(* LS Electric XG5000 project: e_pcmaster_elec_room_controll *)
(* 전기실 환기제어 시스템 실제 적용 시스 템 및 지하주차장 환기 시스탬 *)
(* PLC LSPLC *)
(* module base 0 slot 0: 입출력 모듈:XBC-DR40S (DC 24V 입력 24점, 릴레이 출력 16점) *)
(* module base 0 slot 1: 온도입력 모듈:XBF-RD04A (RTD 온도 입력형 4채널) *)
(* module base 0 slot 2: 아날로그입력 모듈:XBF-AD04A (A/D 전압 전류 입력형 4채널) *)
(* task init: Kind=1 Priority=2 *)
VAR_GLOBAL
    autumn_set_sw : BIT; (* 가을철 온도 *)
    C1_B1_E_FR01_out : BIT;
    C1_B1_E_FR01_start_tk4s_set : WORD;
    C1_B1_E_FR02_out : BIT;
    C1_B1_E_FR02_start_tk4s_set : WORD;
    C1_B1_E_FR05_out : BIT;
    C1_B1_E_FR05_start_tk4s_set : WORD;
    C1_B1_E_FR06_out : BIT;
    C1_B1_E_FR06_start_tk4s_set : WORD;
    C1_B1_E_FR10_out : BIT;
    C1_B1_E_FR10_start_tk4s_set : WORD;
    C1_B1_S_FR03_out : BIT;
    C1_B1_S_FR03_select AT D06230.0 : BIT;
    C1_B1_S_FR03_start_tk4s_alarm_set : WORD;
    C1_B1_S_FR03_temp : WORD;
    C1_B1_S_FR04_out : BIT;
    C1_B1_S_FR04_select AT D06230.1 : BIT;
    C1_B1_S_FR04_start_tk4s_alarm_set : WORD;
    C1_B1_S_FR04_temp : WORD;
    C1_B1_S_FR07_out : BIT;
    C1_B1_S_FR07_select AT D06230.2 : BIT;
    C1_B1_S_FR07_start_tk4s_alarm_set : WORD;
    C1_B1_S_FR07_temp : WORD;
    C1_B1_S_FR08_out : BIT;
    C1_B1_S_FR08_select AT D06230.3 : BIT;
    C1_B1_S_FR08_start_tk4s_alarm_set : WORD;
    C1_B1_S_FR08_temp : WORD;
    C1_B1_S_FR09_out : BIT;
    C1_B1_S_FR09_select AT D06230.4 : BIT;
    C1_B1_S_FR09_start_tk4s_alarm_set : WORD;
    C1_B1_S_FR09_temp : WORD;
    C1_B2_E_FR01_out : BIT;
    C1_B2_E_FR01_start_tk4s_set : WORD;
    C1_B2_E_FR02_out : BIT;
    C1_B2_E_FR02_start_tk4s_set : WORD;
    C1_B2_E_FR05_out : BIT;
    C1_B2_E_FR05_start_tk4s_set : WORD;
    C1_B2_E_FR06_out : BIT;
    C1_B2_E_FR06_start_tk4s_set : WORD;
    C1_B2_E_FR10_out : BIT;
    C1_B2_E_FR10_start_tk4s_set : WORD;
    C1_B2_S_FR03_out : BIT;
    C1_B2_S_FR03_select AT D06230.5 : BIT;
    C1_B2_S_FR03_start_tk4s_alarm_set : WORD;
    C1_B2_S_FR03_temp : WORD;
    C1_B2_S_FR04_out : BIT;
    C1_B2_S_FR04_select AT D06230.6 : BIT;
    C1_B2_S_FR04_start_tk4s_alarm_set : WORD;
    C1_B2_S_FR04_temp : WORD;
    C1_B2_S_FR07_out : BIT;
    C1_B2_S_FR07_select AT D06230.7 : BIT;
    C1_B2_S_FR07_start_tk4s_alarm_set : WORD;
    C1_B2_S_FR07_temp : WORD;
    C1_B2_S_FR08_out : BIT;
    C1_B2_S_FR08_select AT D06230.8 : BIT;
    C1_B2_S_FR08_start_tk4s_alarm_set : WORD;
    C1_B2_S_FR08_temp : WORD;
    C1_B2_S_FR09_out : BIT;
    C1_B2_S_FR09_select AT D06230.9 : BIT;
    C1_B2_S_FR09_start_tk4s_alarm_set : WORD;
    C1_B2_S_FR09_temp : WORD;
    C2_B1_E_FR11_out : BIT;
    C2_B1_E_FR11_start_tk4s_set : WORD;
    C2_B1_S_FR12_out : BIT;
    C2_B1_S_FR12_select AT D06230.A : BIT;
    C2_B1_S_FR12_start_tk4s_alarm_set : WORD;
    C2_B1_S_FR12_temp : WORD;
    C2_B2_E_FR11_out : BIT;
    C2_B2_E_FR11_start_tk4s_set : WORD;
    C2_B2_S_FR12_out : BIT;
    C2_B2_S_FR12_select AT D06230.B : BIT;
    C2_B2_S_FR12_start_tk4s_alarm_set : WORD;
    C2_B2_S_FR12_temp : WORD;
    C2_B3_E_FR11_out : BIT;
    C2_B3_E_FR11_start_tk4s_set : WORD;
    C2_B3_S_FR12_out : BIT;
    C2_B3_S_FR12_select AT D06230.C : BIT;
    C2_B3_S_FR12_start_tk4s_alarm_set : WORD;
    C2_B3_S_FR12_temp : WORD;
    cold_winter_set_sw : BIT;
    early_winter_set_sw : BIT; (* 초겨울 *)
    EF_operation AT M00203 : BIT;
    heart_beat_manual_sw : BIT;
    heart_beat_mem : WORD;
    heart_beat_timer : TIMER;
    Park_1H_time : WORD;
    Park_auto_B_manual_A : BIT;
    Park_auto_start : BIT;
    Park_daily_schedule_on : BIT;
    Park_manual_cont_ind_start : BIT;
    Park_manual_cont_tot_start : BIT;
    Park_manual_con_B_time_A : BIT;
    Park_manual_ind_B_tot_A : BIT;
    Park_manual_ind_start_out : BIT;
    Park_manual_oper_time : WORD;
    Park_manual_start : BIT;
    Park_manual_timer : TIMER;
    Park_manual_time_ind_start : BIT;
    Park_manual_time_tot_start : BIT;
    Park_manual_total_start_out : BIT;
    Park_manual_순차가동_2R : DWORD;
    Park_manual_순차기동_계산값 : WORD;
    Park_manual_순차기동_전송값 : WORD;
    Park_schedule_06_start : BIT;
    Park_schedule_08_start : BIT;
    Park_schedule_09_start : BIT;
    Park_schedule_10_start : BIT;
    Park_schedule_15_stop : BIT;
    Park_schedule_17stop : BIT;
    Park_schedule_18stop : BIT;
    Park_schedule_20stop : BIT;
    Park_schedule_autumn : BIT;
    Park_schedule_spring : BIT;
    Park_schedule_summer : BIT;
    Park_schedule_winter : BIT;
    Park_start_B_stop_A : BIT;
    Park_temp_1_high : WORD;
    Park_temp_1_high_H_set : WORD;
    Park_temp_1_high_L_set : WORD;
    Park_temp_2_med_high : WORD;
    Park_temp_2_med_high_H_set : WORD;
    Park_temp_2_med_high_L_set : WORD;
    Park_temp_3_med : WORD;
    Park_temp_3_med_H_set : WORD;
    Park_temp_3_med_L_set : WORD;
    Park_temp_4_med_low : WORD;
    Park_temp_4_med_low_H_set : WORD;
    Park_temp_4_med_low_L_set : WORD;
    Park_temp_5_low : WORD;
    Park_temp_5_low_H_set : WORD;
    Park_temp_5_low_L_set : WORD;
    Park_temp_6_low_1 : WORD;
    Park_temp_6_low_1_oper_time : WORD;
    Park_temp_7_low_2 : WORD;
    Park_temp_7_low_2_oper_time : WORD;
    Park_temp_8_low_3 : WORD;
    Park_temp_8_low_3_oper_time : WORD;
    Park_temp_9_below0 : WORD;
    Park_temp_9_below0_oper_time : WORD;
    Park_time_oper_delay_time : WORD;
    Park_tk4m_alarm_start_set : WORD;
    Park_tk4m_alarm_stop_set : WORD;
    Park_tk4m_start_set : WORD;
    Park_tk4m_stop_set : WORD;
    Park_순차기동_카운터 : COUNTER;
    Park_순차기동_타이머 : TIMER;
    SF_operation AT M00209 : BIT;
    spring_set_sw : BIT; (* spring_set_sw *)
    summer_set_sw : BIT; (* 하절기운전온도 변경 *)
    tr01_1m_high_temp_from_pc AT D00980 : WORD;
    tr01_temp_scaled_value AT D00024 : WORD;
    tr02_1m_high_temp_from_pc AT D00981 : WORD;
    tr02_temp_scaled_value AT D00025 : WORD;
    tr03_1m_high_temp_from_pc AT D00982 : WORD;
    tr03_temp_scaled_value AT D00026 : WORD;
    winter_set_sw : BIT; (* 겨울철 *)
    _002_1C_1B_FR01_temp : WORD; (* _002_1C_1B_FR01_temp *)
    _002_1C_1B_FR02_temp : WORD; (* _002_1C_1B_FR02_temp *)
    _002_1C_1B_FR03_temp : WORD; (* _002_1C_1B_FR03_temp *)
    _002_1C_1B_FR04_temp : WORD; (* _002_1C_1B_FR04_temp *)
    _002_1C_1B_FR05_temp : WORD; (* _002_1C_1B_FR05_temp *)
    _002_1C_2B_FR01_temp : WORD; (* _002_1C_2B_FR01_temp *)
    _002_1C_2B_FR02_temp : WORD; (* _002_1C_2B_FR02_temp *)
    _002_1C_2B_FR03_temp : WORD; (* _002_1C_2B_FR03_temp *)
    _002_1C_2B_FR04_temp : WORD; (* _002_1C_2B_FR04_temp *)
    _002_1C_2B_FR05_temp : WORD; (* _002_1C_2B_FR05_temp *)
    _002_tr_1_temp : WORD; (* _002_tr_1_temp *)
    _002_tr_2_temp : WORD; (* _002_tr_2_temp *)
    _002_tr_3_temp : WORD; (* _002_tr_3_temp *)
    _002_W_011_reserved : WORD; (* _002_W_011_reserved *)
    _002_W_012_reserved : WORD; (* _002_W_012_reserved *)
    _003_tr_1_AB_valtage : DWORD; (* _003_tr_1_AB_valtage *)
    _003_tr_1_A_current : DWORD; (* _003_tr_1_A_current *)
    _003_tr_1_A_valtage : DWORD; (* _003_tr_1_A_valtage *)
    _003_tr_1_BC_valtage : DWORD; (* _003_tr_1_BC_valtage *)
    _003_tr_1_B_current : DWORD; (* _003_tr_1_B_current *)
    _003_tr_1_B_valtage : DWORD; (* _003_tr_1_B_valtage *)
    _003_tr_1_CA_valtage : DWORD; (* _003_tr_1_CA_valtage *)
    _003_tr_1_C_current : DWORD; (* _003_tr_1_C_current *)
    _003_tr_1_C_valtage : DWORD; (* _003_tr_1_C_valtage *)
    _003_tr_1_effective_power : DWORD; (* _003_tr_1_effective_power *)
    _003_tr_1_power : DWORD; (* _003_tr_1_power *)
    _003_tr_1_power_factor : DWORD; (* _003_tr_1_power_factor *)
    _003_tr_1_reactive_power : DWORD; (* _003_tr_1_reactive_power *)
    _004_tr_2_AB_valtage : DWORD; (* _004_tr_2_AB_valtage *)
    _004_tr_2_A_current : DWORD; (* _004_tr_2_A_current *)
    _004_tr_2_A_valtage : DWORD; (* _004_tr_2_A_valtage *)
    _004_tr_2_BC_valtage : DWORD; (* _004_tr_2_BC_valtage *)
    _004_tr_2_B_current : DWORD; (* _004_tr_2_B_current *)
    _004_tr_2_B_valtage : DWORD; (* _004_tr_2_B_valtage *)
    _004_tr_2_CA_valtage : DWORD; (* _004_tr_2_CA_valtage *)
    _004_tr_2_C_current : DWORD; (* _004_tr_2_C_current *)
    _004_tr_2_C_valtage : DWORD; (* _004_tr_2_C_valtage *)
    _004_tr_2_effective_power : DWORD; (* _004_tr_2_effective_power *)
    _004_tr_2_power : DWORD; (* _004_tr_2_power *)
    _004_tr_2_power_factor : DWORD; (* _004_tr_2_power_factor *)
    _004_tr_2_reactive_power : DWORD; (* _004_tr_2_reactive_power *)
    _005_tr_3_AB_valtage : DWORD; (* _005_tr_3_AB_valtage *)
    _005_tr_3_A_current : DWORD; (* _005_tr_3_A_current *)
    _005_tr_3_A_valtage : DWORD; (* _005_tr_3_A_valtage *)
    _005_tr_3_BC_valtage : DWORD; (* _005_tr_3_BC_valtage *)
    _005_tr_3_B_current : DWORD; (* _005_tr_3_B_current *)
    _005_tr_3_B_valtage : DWORD; (* _005_tr_3_B_valtage *)
    _005_tr_3_CA_valtage : DWORD; (* _005_tr_3_CA_valtage *)
    _005_tr_3_C_current : DWORD; (* _005_tr_3_C_current *)
    _005_tr_3_C_valtage : DWORD; (* _005_tr_3_C_valtage *)
    _005_tr_3_effective_power : DWORD; (* _005_tr_3_effective_power *)
    _005_tr_3_power : DWORD; (* _005_tr_3_power *)
    _005_tr_3_power_factor : DWORD; (* _005_tr_3_power_factor *)
    _005_tr_3_reactive_power : DWORD; (* _005_tr_3_reactive_power *)
    _007_outdoor_temp : WORD; (* _007_outdoor_temp *)
    _007_room_temp : WORD; (* _007_room_temp *)
    _008_room_temp_high_set AT D00906 : WORD; (* _008_room_temp_high_set *)
    _008_room_temp_high_set_high_limit : WORD; (* _008_room_temp_high_set_high_limit *)
    _008_room_temp_high_set_low_limit : WORD; (* _008_room_temp_high_set_low_limit *)
    _008_room_temp_low_set AT D00907 : WORD; (* _008_room_temp_low_set *)
    _008_room_temp_low_set_high_limit : WORD; (* _008_room_temp_low_set_high_limit *)
    _008_room_temp_low_set_low_limit : WORD; (* _008_room_temp_low_set_low_limit *)
    _009_outdoor_temp_high_set AT D00908 : WORD; (* _009_outdoor_temp_high_set *)
    _009_outdoor_temp_high_set_high_limit : WORD; (* _009_outdoor_temp_high_set_high_limit *)
    _009_outdoor_temp_high_set_low_limit : WORD; (* _009_outdoor_temp_high_set_low_limit *)
    _009_outdoor_temp_low_set AT D00909 : WORD; (* _009_outdoor_temp_low_set *)
    _009_outdoor_temp_low_set_high_limit : WORD; (* _009_outdoor_temp_low_set_high_limit *)
    _009_outdoor_temp_low_set_low_limit : WORD; (* _009_outdoor_temp_low_set_low_limit *)
    _010_D_00 : DWORD; (* _010_D_00 *)
    _010_D_01 : DWORD; (* _010_D_01 *)
    _010_D_unit_hour_cost : DWORD; (* _010_D_unit_hour_cost *)
    _010_R_00 : DWORD; (* _010_R_00 *)
    _010_R_01 : DWORD; (* _010_R_01 *)
    _010_R_power_unit_price_percent : DWORD; (* _010_R_power_unit_price_percent *)
    _010_R_unit_hour_cost : DWORD; (* _010_R_unit_hour_cost *)
    _010_W_02 : WORD; (* _010_W_02 *)
    _010_W_03 : WORD; (* _010_W_03 *)
    _010_W_1hr_count : WORD; (* _010_W_1hr_count *)
    _010_W_1_thousand_hour : WORD; (* _010_W_1_thousand_hour *)
    _010_W_fan_power_capacity : WORD; (* _010_W_fan_power_capacity *)
    _010_W_high_low_diff : WORD; (* _010_W_high_low_diff *)
    _010_W_power_unit_price : WORD; (* _010_W_power_unit_price *)
    _010_W_TR1_temp_high_set AT D00900 : WORD;
    _010_W_TR1_temp_low_set AT D00901 : WORD;
    _010_W_TR2_temp_high_set AT D00902 : WORD;
    _010_W_TR2_temp_low_set AT D00903 : WORD;
    _010_W_TR3_temp_high_set AT D00904 : WORD; (* _010_W_TR_temp_high_set *)
    _010_W_TR3_temp_low_set AT D00905 : WORD; (* _010_W_TR_temp_low_set *)
    _01_CH0_TEMP AT U01.04 : WORD; (* 온도입력모듈 : 채널0 온도변환값(전기실온도) *)
    _01_CH1_TEMP AT U01.05 : WORD; (* 온도입력모듈 : 채널1 온도변환값(외기온도) *)
    _01_CH2_TEMP AT U01.06 : WORD; (* 온도입력모듈 : 채널2 온도변환값(에어콘01출구온도) *)
    _01_CH3_TEMP AT U01.07 : WORD; (* 온도입력모듈 : 채널3 온도변환값(에어콘02출구온도) *)
    _02_CH0_DATA AT U02.02 : WORD; (* 아날로그입력 모듈: 채널0 변환값(tr01 temp) *)
    _02_CH1_DATA AT U02.03 : WORD; (* 아날로그입력 모듈: 채널1 변환값(tr02 temp) *)
    _02_CH2_DATA AT U02.04 : WORD; (* 아날로그입력 모듈: 채널2 변환값(tr01 temp) *)
    _IC_1B_FR01_temp_high_set : BIT;
    _주차장_급기팬_가동 : BIT;
    _주차장_급기팬_정지 : BIT;
    월간타이머리셋 : BIT;
    전기실_급배기_동시기동방지 : TIMER; (* 전기실_급배기_동시기동방지 *)
    주차장_급기가동온도 : WORD;
    주차장_급기정지온도 : WORD; (* 주차장_제어_외기_고온도 *)
END_VAR
VAR_GLOBAL RETAIN
    Park_oper_time_add : WORD;
    TR1_opertime_time : WORD;
    TR1_opertime_timer : TIMER;
    TR2_opertime_time : WORD;
    TR2_opertime_timer : TIMER;
    TR3_opertime_time : WORD;
    TR3_opertime_timer : TIMER;
    TR_opertime_total_time : WORD;
    _000_EF_tot_local_auto_op_timer : TIMER; (* _000_EF_tot_local_auto_op_timer *)
    _000_EF_tot_local_manual_op_timer : TIMER; (* _000_EF_tot_local_manual_op_timer *)
    _000_EF_tot_op_room_op_timer : TIMER; (* _000_EF_tot_op_room_op_timer *)
    _000_EF_tot_op_timer : TIMER; (* _000_EF_tot_op_timer *)
    _000_SF_tot_local_auto_op_timer : TIMER; (* _000_SF_tot_local_auto_op_timer *)
    _000_SF_tot_local_manual_op_timer : TIMER; (* _000_SF_tot_local_manual_op_timer *)
    _000_SF_tot_op_room_op_timer : TIMER; (* _000_SF_tot_op_room_op_timer *)
    _000_SF_tot_op_timer : TIMER; (* _000_SF_tot_op_timer *)
    _001_EF_tot_local_auto_op_hour : WORD; (* _001_EF_tot_local_auto_op_hour *)
    _001_EF_tot_local_manual_op_hour : WORD; (* _001_EF_tot_local_manual_op_hour *)
    _001_EF_tot_op_hour : WORD; (* _001_EF_tot_op_hour *)
    _001_EF_tot_op_room_op_hour : WORD; (* _001_EF_tot_op_room_op_hour *)
    _001_SF_tot_local_auto_op_hour : WORD; (* _001_SF_tot_local_auto_op_hour *)
    _001_SF_tot_local_manual_op_hour : WORD; (* _001_SF_tot_local_manual_op_hour *)
    _001_SF_tot_op_hour : WORD; (* _001_SF_tot_op_hour *)
    _001_SF_tot_op_room_op_hour : WORD; (* _001_SF_tot_op_room_op_hour *)
    _001_tot_local_auto_op_hour : WORD; (* _001_tot_local_auto_op_hour *)
    _001_tot_local_manual_op_hour : WORD; (* _001_tot_local_manual_op_hour *)
    _001_tot_op_hour : WORD; (* _001_tot_op_hour *)
    _001_tot_op_room_op_hour : WORD; (* _001_tot_op_room_op_hour *)
    _006_EF_tot_local_auto_op_hour : COUNTER; (* _006_EF_tot_local_auto_op_hour *)
    _006_EF_tot_local_manual_op_hour : COUNTER; (* _006_EF_tot_local_manual_op_hour *)
    _006_EF_tot_op_hour : COUNTER; (* _006_ESF_tot_op_hour *)
    _006_EF_tot_op_room_op_hour : COUNTER; (* _006_EF_tot_op_room_op_hour *)
    _006_SF_tot_local_auto_op_hour : COUNTER; (* _006_SF_tot_local_auto_op_hour *)
    _006_SF_tot_local_manual_op_hour : COUNTER; (* _006_SF_tot_local_manual_op_hour *)
    _006_SF_tot_op_hour : COUNTER; (* _006_SF_tot_op_hour *)
    _006_SF_tot_op_room_op_hour : COUNTER; (* _006_SF_tot_op_room_op_hour *)
END_VAR

PROGRAM elec_room_ventilation (* task: 스캔 프로그램 *)
VAR
    aircon01_operation AT M00221 : BIT;
    aircon01_OP_value AT D00957 : WORD;
    aircon02_operation AT M00222 : BIT;
    aircon02_OP_value AT D00958 : WORD;
    aircon_operation : BIT;
    basic_win_2_main_menu : BIT; (* basic_win_2_main_menu *)
    basic_win_2_main_menu_action : BIT; (* basic_win_2_main_menu_action *)
    basic_win_3_main_menu : BIT; (* basic_win_3_main_menu *)
    basic_win_3_main_menu_action : BIT; (* basic_win_3_main_menu_action *)
    basic_win_5_main_menu : BIT; (* basic_win_5_main_menu *)
    basic_win_5_main_menu_action : BIT; (* basic_win_5_main_menu_action *)
    EF_local_auto_start AT M00105 : BIT; (* EF_local_auto_start *)
    EF_local_auto_start_out AT M00200 : BIT; (* EF_local_auto_start_out *)
    EF_local_manual_start AT M00106 : BIT; (* EF_local_manual_start *)
    EF_local_manual_start_out AT M00201 : BIT; (* EF_local_manual_start_out *)
    EF_local_manual_start_sw AT M00116 : BIT; (* EF_local_manual_start_sw *)
    EF_op_room_start AT M00107 : BIT; (* EF_op_room_start *)
    EF_op_room_start_out AT M00202 : BIT; (* EF_op_room_start_out *)
    EF_stop AT M00108 : BIT; (* EF_stop *)
    EF_stop_out AT M00204 : BIT; (* EF_stop_out *)
    EF_trip AT M00205 : BIT; (* EF_trip *)
    EF_trip_reset AT M00109 : BIT; (* EF_trip_reset *)
    outdoor_temp_high_set_sw : BIT; (* outdoor_temp_high_set_sw *)
    outdoor_temp_low_set_sw : BIT; (* outdoor_temp_low_set_sw *)
    plc_error : BIT;
    plc_run : BIT;
    room_temp_high_set_sw : BIT; (* room_temp_high_set_sw *)
    room_temp_low_set_sw : BIT; (* room_temp_low_set_sw *)
    room_temp_trend_win_open : BIT; (* room_temp_trend_win_open *)
    room_temp_trend_win_trigger : BIT; (* room_temp_trend_win_trigger *)
    SF_local_auto_point_hour : BIT; (* SF_local_auto_point_hour *)
    SF_local_auto_start AT M00110 : BIT; (* SF_local_auto_start *)
    SF_local_auto_start_out AT M00206 : BIT; (* SF_local_auto_start_out *)
    SF_local_manual_point_hour : BIT; (* SF_local_manual_point_hour *)
    SF_local_manual_start AT M00111 : BIT; (* SF_local_manual_start *)
    SF_local_manual_start_out AT M00207 : BIT; (* SF_local_manual_start_out *)
    SF_local_manual_start_sw AT M00117 : BIT; (* SF_local_manual_start_sw *)
    SF_op_room_point_hour : BIT; (* SF_op_room_point_hour *)
    SF_op_room_start AT M00112 : BIT; (* SF_op_room_start *)
    SF_op_room_start_out AT M00208 : BIT; (* SF_op_room_start_out *)
    SF_stop AT M00113 : BIT; (* SF_stop *)
    SF_stop_out AT M00210 : BIT; (* SF_stop_out *)
    SF_tot_point_hour : BIT; (* SF_tot_point_hour *)
    sf_trip AT M00211 : BIT; (* sf_trip *)
    SF_trip_reset AT M00114 : BIT; (* SF_trip_reset *)
    tr_temp_trend_win_open : BIT; (* tr_temp_trend_win_open *)
    tr_temp_trend_win_trigger : BIT; (* tr_temp_trend_win_trigger *)
    unit_price_change : BIT; (* unit_price_change *)
    unit_price_change_action : BIT; (* unit_price_change_action *)
    unit_price_change_complete : BIT; (* unit_price_change_complete *)
    unit_price_change_complete_action : BIT; (* unit_price_change_complete_action *)
    unit_price_change_password : WORD; (* unit_price_change_password *)
    unit_price_change_password_fail : BIT; (* unit_price_change_password_fail *)
    unit_price_change_password_ok : BIT; (* unit_price_change_password_ok *)
    unit_price_change_pw_fail : BIT; (* unit_price_change_pw_fail *)
    unit_price_change_pw_ok : BIT; (* unit_price_change_pw_ok *)
    unit_price_change_temp_value : WORD; (* unit_price_change_temp_value *)
    win_2_view_graph : BIT; (* win_2_view_graph *)
    win_2_view_graph_open : BIT; (* win_2_view_graph_open *)
    _007_outdoor_temp_max_reset : BIT;
END_VAR
VAR_EXTERNAL
    autumn_set_sw : BIT; (* 가을철 온도 *)
    EF_operation : BIT; (* AT M00203 *)
    heart_beat_manual_sw : BIT;
    heart_beat_mem : WORD;
    heart_beat_timer : TIMER;
    SF_operation : BIT; (* AT M00209 *)
    tr01_1m_high_temp_from_pc : WORD; (* AT D00980 *)
    tr01_temp_scaled_value : WORD; (* AT D00024 *)
    tr02_1m_high_temp_from_pc : WORD; (* AT D00981 *)
    tr02_temp_scaled_value : WORD; (* AT D00025 *)
    tr03_1m_high_temp_from_pc : WORD; (* AT D00982 *)
    tr03_temp_scaled_value : WORD; (* AT D00026 *)
    winter_set_sw : BIT; (* 겨울철 *)
    _007_outdoor_temp : WORD; (* _007_outdoor_temp *)
    _007_room_temp : WORD; (* _007_room_temp *)
    _008_room_temp_high_set : WORD; (* AT D00906 *) (* _008_room_temp_high_set *)
    _008_room_temp_high_set_high_limit : WORD; (* _008_room_temp_high_set_high_limit *)
    _008_room_temp_high_set_low_limit : WORD; (* _008_room_temp_high_set_low_limit *)
    _008_room_temp_low_set : WORD; (* AT D00907 *) (* _008_room_temp_low_set *)
    _008_room_temp_low_set_high_limit : WORD; (* _008_room_temp_low_set_high_limit *)
    _008_room_temp_low_set_low_limit : WORD; (* _008_room_temp_low_set_low_limit *)
    _009_outdoor_temp_high_set : WORD; (* AT D00908 *) (* _009_outdoor_temp_high_set *)
    _009_outdoor_temp_low_set : WORD; (* AT D00909 *) (* _009_outdoor_temp_low_set *)
    _010_W_power_unit_price : WORD; (* _010_W_power_unit_price *)
    _01_CH0_TEMP : WORD; (* AT U01.04 *) (* 온도입력모듈 : 채널0 온도변환값(전기실온도) *)
    _01_CH1_TEMP : WORD; (* AT U01.05 *) (* 온도입력모듈 : 채널1 온도변환값(외기온도) *)
    월간타이머리셋 : BIT;
    전기실_급배기_동시기동방지 : TIMER; (* 전기실_급배기_동시기동방지 *)
END_VAR

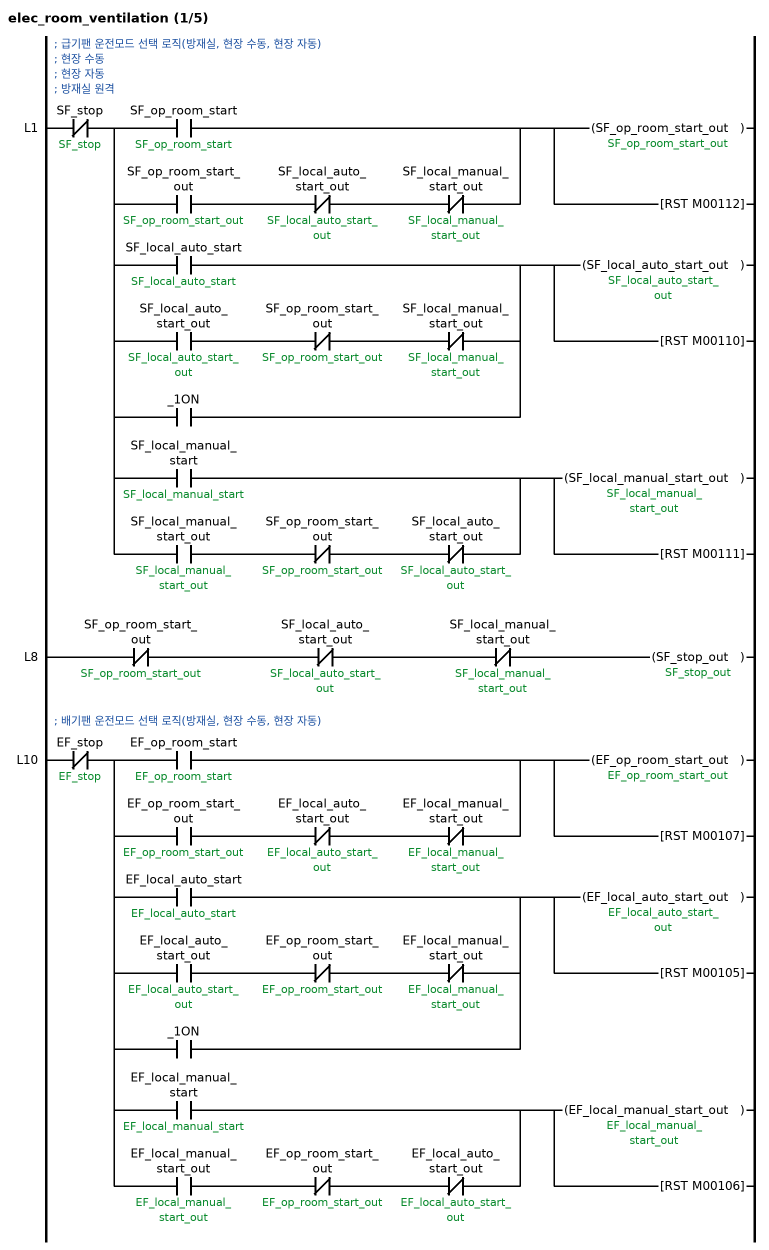
// 급기팬 운전모드 선택 로직(방재실, 현장 수동, 현장 자동)
; L1
LOAD NOT  SF_stop	// SF_stop
MPUSH
LOAD      SF_op_room_start	// SF_op_room_start
LOAD      SF_op_room_start_out	// SF_op_room_start_out
AND NOT   SF_local_auto_start_out	// SF_local_auto_start_out
AND NOT   SF_local_manual_start_out	// SF_local_manual_start_out
OR LOAD
AND LOAD
OUT       SF_op_room_start_out	// SF_op_room_start_out
RST       M00112
MLOAD
LOAD      SF_local_auto_start	// SF_local_auto_start
LOAD      SF_local_auto_start_out	// SF_local_auto_start_out
AND NOT   SF_op_room_start_out	// SF_op_room_start_out
AND NOT   SF_local_manual_start_out	// SF_local_manual_start_out
OR LOAD
OR        _1ON
AND LOAD
OUT       SF_local_auto_start_out	// SF_local_auto_start_out
RST       M00110
MPOP
LOAD      SF_local_manual_start	// SF_local_manual_start
LOAD      SF_local_manual_start_out	// SF_local_manual_start_out
AND NOT   SF_op_room_start_out	// SF_op_room_start_out
AND NOT   SF_local_auto_start_out	// SF_local_auto_start_out
OR LOAD
AND LOAD
OUT       SF_local_manual_start_out	// SF_local_manual_start_out
RST       M00111
// output comment: 현장 수동
// output comment: 현장 자동
// output comment: 방재실 원격
; L8
LOAD NOT  SF_op_room_start_out	// SF_op_room_start_out
AND NOT   SF_local_auto_start_out	// SF_local_auto_start_out
AND NOT   SF_local_manual_start_out	// SF_local_manual_start_out
OUT       SF_stop_out	// SF_stop_out
// 배기팬 운전모드 선택 로직(방재실, 현장 수동, 현장 자동)
; L10
LOAD NOT  EF_stop	// EF_stop
MPUSH
LOAD      EF_op_room_start	// EF_op_room_start
LOAD      EF_op_room_start_out	// EF_op_room_start_out
AND NOT   EF_local_auto_start_out	// EF_local_auto_start_out
AND NOT   EF_local_manual_start_out	// EF_local_manual_start_out
OR LOAD
AND LOAD
OUT       EF_op_room_start_out	// EF_op_room_start_out
RST       M00107
MLOAD
LOAD      EF_local_auto_start	// EF_local_auto_start
LOAD      EF_local_auto_start_out	// EF_local_auto_start_out
AND NOT   EF_op_room_start_out	// EF_op_room_start_out
AND NOT   EF_local_manual_start_out	// EF_local_manual_start_out
OR LOAD
OR        _1ON
AND LOAD
OUT       EF_local_auto_start_out	// EF_local_auto_start_out
RST       M00105
MPOP
LOAD      EF_local_manual_start	// EF_local_manual_start
LOAD      EF_local_manual_start_out	// EF_local_manual_start_out
AND NOT   EF_op_room_start_out	// EF_op_room_start_out
AND NOT   EF_local_auto_start_out	// EF_local_auto_start_out
OR LOAD
AND LOAD
OUT       EF_local_manual_start_out	// EF_local_manual_start_out
RST       M00106

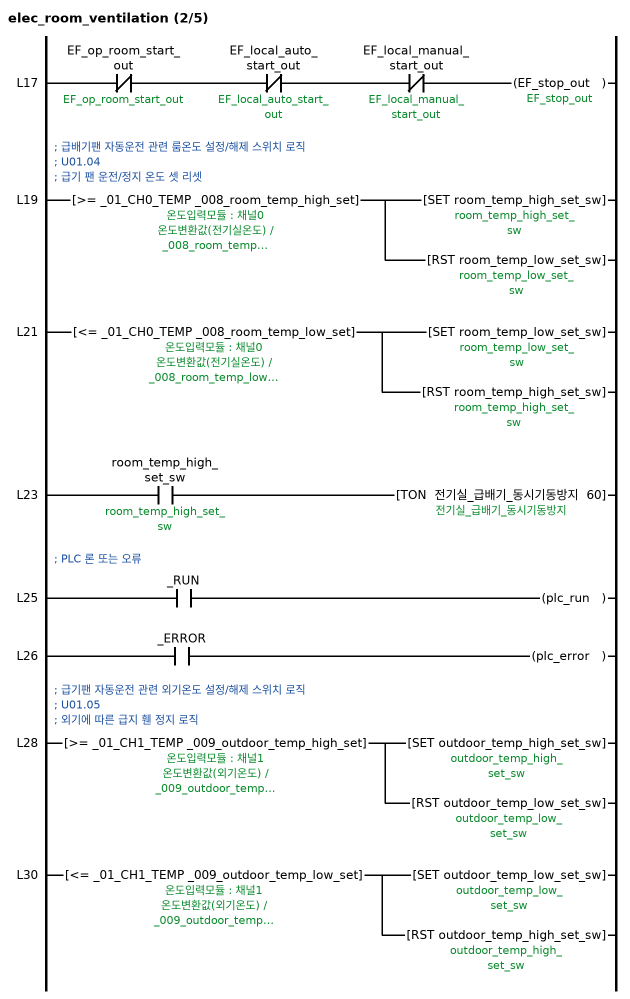
; L17
LOAD NOT  EF_op_room_start_out	// EF_op_room_start_out
AND NOT   EF_local_auto_start_out	// EF_local_auto_start_out
AND NOT   EF_local_manual_start_out	// EF_local_manual_start_out
OUT       EF_stop_out	// EF_stop_out
// 급배기팬 자동운전 관련 룸온도 설정/해제 스위치 로직
; L19
LOAD>=    _01_CH0_TEMP _008_room_temp_high_set	// 온도입력모듈 : 채널0 온도변환값(전기실온도) / _008_room_temp_high_set
SET       room_temp_high_set_sw	// room_temp_high_set_sw
RST       room_temp_low_set_sw	// room_temp_low_set_sw
// output comment: U01.04
// output comment: 급기 팬 운전/정지 온도 셋 리셋
; L21
LOAD<=    _01_CH0_TEMP _008_room_temp_low_set	// 온도입력모듈 : 채널0 온도변환값(전기실온도) / _008_room_temp_low_set
SET       room_temp_low_set_sw	// room_temp_low_set_sw
RST       room_temp_high_set_sw	// room_temp_high_set_sw
; L23
LOAD      room_temp_high_set_sw	// room_temp_high_set_sw
TON       전기실_급배기_동시기동방지 60	// 전기실_급배기_동시기동방지
// PLC 론 또는 오류
; L25
LOAD      _RUN
OUT       plc_run
; L26
LOAD      _ERROR
OUT       plc_error
// 급기팬 자동운전 관련 외기온도 설정/해제 스위치 로직
; L28
LOAD>=    _01_CH1_TEMP _009_outdoor_temp_high_set	// 온도입력모듈 : 채널1 온도변환값(외기온도) / _009_outdoor_temp_high_set
SET       outdoor_temp_high_set_sw	// outdoor_temp_high_set_sw
RST       outdoor_temp_low_set_sw	// outdoor_temp_low_set_sw
// output comment: U01.05
// output comment: 외기에 따른 급지 휀 정지 로직
; L30
LOAD<=    _01_CH1_TEMP _009_outdoor_temp_low_set	// 온도입력모듈 : 채널1 온도변환값(외기온도) / _009_outdoor_temp_low_set
SET       outdoor_temp_low_set_sw	// outdoor_temp_low_set_sw
RST       outdoor_temp_high_set_sw	// outdoor_temp_high_set_sw

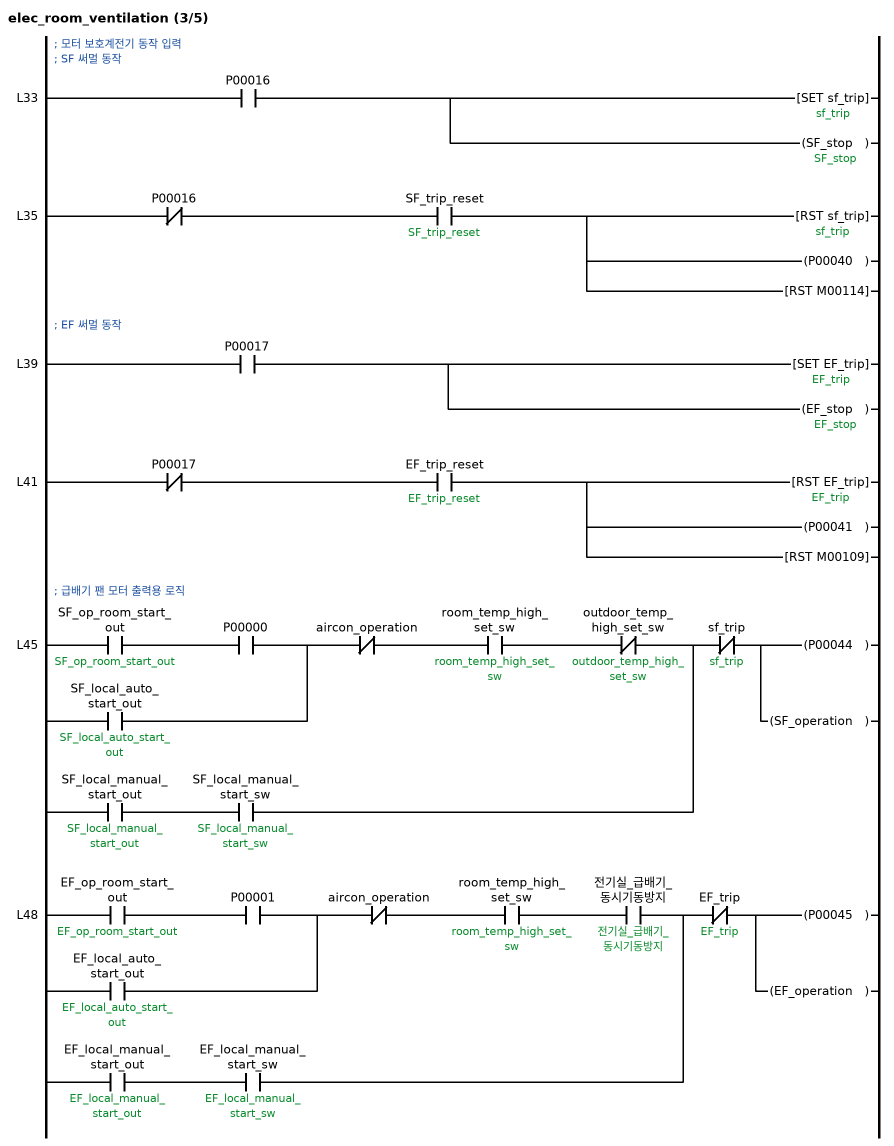
// 모터 보호계전기 동작 입력
; L33
LOAD      P00016
SET       sf_trip	// sf_trip
OUT       SF_stop	// SF_stop
// output comment: SF 써멀 동작
; L35
LOAD NOT  P00016
AND       SF_trip_reset	// SF_trip_reset
RST       sf_trip	// sf_trip
OUT       P00040
RST       M00114
; L39
LOAD      P00017
SET       EF_trip	// EF_trip
OUT       EF_stop	// EF_stop
// output comment: EF 써멀 동작
; L41
LOAD NOT  P00017
AND       EF_trip_reset	// EF_trip_reset
RST       EF_trip	// EF_trip
OUT       P00041
RST       M00109
// 급배기 팬 모터 출력용 로직
; L45
LOAD      SF_op_room_start_out	// SF_op_room_start_out
AND       P00000
OR        SF_local_auto_start_out	// SF_local_auto_start_out
AND NOT   aircon_operation
AND       room_temp_high_set_sw	// room_temp_high_set_sw
AND NOT   outdoor_temp_high_set_sw	// outdoor_temp_high_set_sw
LOAD      SF_local_manual_start_out	// SF_local_manual_start_out
AND       SF_local_manual_start_sw	// SF_local_manual_start_sw
OR LOAD
AND NOT   sf_trip	// sf_trip
OUT       P00044
OUT       SF_operation
; L48
LOAD      EF_op_room_start_out	// EF_op_room_start_out
AND       P00001
OR        EF_local_auto_start_out	// EF_local_auto_start_out
AND NOT   aircon_operation
AND       room_temp_high_set_sw	// room_temp_high_set_sw
AND       전기실_급배기_동시기동방지	// 전기실_급배기_동시기동방지
LOAD      EF_local_manual_start_out	// EF_local_manual_start_out
AND       EF_local_manual_start_sw	// EF_local_manual_start_sw
OR LOAD
AND NOT   EF_trip	// EF_trip
OUT       P00045
OUT       EF_operation

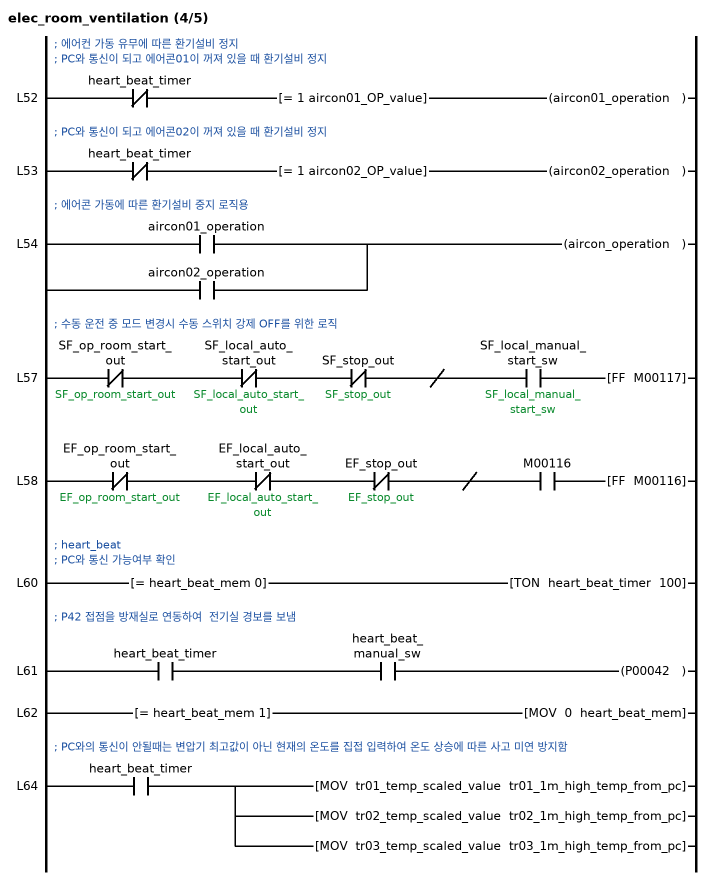
// 에어컨 가동 유무에 따른 환기설비 정지
; L52
LOAD NOT  heart_beat_timer
AND=      1 aircon01_OP_value
OUT       aircon01_operation
// output comment: PC와 통신이 되고 에어콘01이 꺼져 있을 때 환기설비 정지
; L53
LOAD NOT  heart_beat_timer
AND=      1 aircon02_OP_value
OUT       aircon02_operation
// output comment: PC와 통신이 되고 에어콘02이 꺼져 있을 때 환기설비 정지
; L54
LOAD      aircon01_operation
OR        aircon02_operation
OUT       aircon_operation
// output comment: 에어콘 가동에 따른 환기설비 중지 로직용
// 수동 운전 중 모드 변경시 수동 스위치 강제 OFF를 위한 로직
; L57
LOAD NOT  SF_op_room_start_out	// SF_op_room_start_out
AND NOT   SF_local_auto_start_out	// SF_local_auto_start_out
AND NOT   SF_stop_out	// SF_stop_out
NOT
AND       SF_local_manual_start_sw	// SF_local_manual_start_sw
FF        M00117
; L58
LOAD NOT  EF_op_room_start_out	// EF_op_room_start_out
AND NOT   EF_local_auto_start_out	// EF_local_auto_start_out
AND NOT   EF_stop_out	// EF_stop_out
NOT
AND       M00116
FF        M00116
// heart_beat
; L60
LOAD=     heart_beat_mem 0
TON       heart_beat_timer 100
// output comment: PC와 통신 가능여부 확인
; L61
LOAD      heart_beat_timer
AND       heart_beat_manual_sw
OUT       P00042
// output comment: P42 접점을 방재실로 연동하여  전기실 경보를 보냄
; L62
LOAD=     heart_beat_mem 1
MOV       0 heart_beat_mem
; L64
LOAD      heart_beat_timer
MOV       tr01_temp_scaled_value tr01_1m_high_temp_from_pc
MOV       tr02_temp_scaled_value tr02_1m_high_temp_from_pc
MOV       tr03_temp_scaled_value tr03_1m_high_temp_from_pc
// output comment: PC와의 통신이 안될때는 변압기 최고값이 아닌 현재의 온도를 집접 입력하여 온도 상승에 따른 사고 미연 방지함

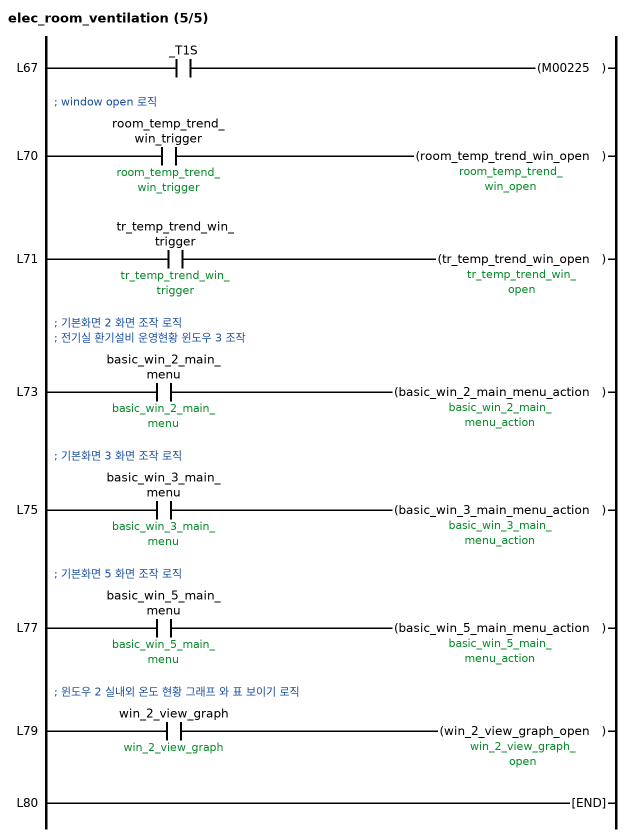
; L67
LOAD      _T1S
OUT       M00225
// window open 로직
; L70
LOAD      room_temp_trend_win_trigger	// room_temp_trend_win_trigger
OUT       room_temp_trend_win_open	// room_temp_trend_win_open
; L71
LOAD      tr_temp_trend_win_trigger	// tr_temp_trend_win_trigger
OUT       tr_temp_trend_win_open	// tr_temp_trend_win_open
// 기본화면 2 화면 조작 로직
; L73
LOAD      basic_win_2_main_menu	// basic_win_2_main_menu
OUT       basic_win_2_main_menu_action	// basic_win_2_main_menu_action
// output comment: 전기실 환기설비 운영현황 윈도우 3 조작
// 기본화면 3 화면 조작 로직
; L75
LOAD      basic_win_3_main_menu	// basic_win_3_main_menu
OUT       basic_win_3_main_menu_action	// basic_win_3_main_menu_action
// 기본화면 5 화면 조작 로직
; L77
LOAD      basic_win_5_main_menu	// basic_win_5_main_menu
OUT       basic_win_5_main_menu_action	// basic_win_5_main_menu_action
// 윈도우 2 실내외 온도 현황 그래프 와 표 보이기 로직
; L79
LOAD      win_2_view_graph	// win_2_view_graph
OUT       win_2_view_graph_open	// win_2_view_graph_open
; L80
END
END_PROGRAM

PROGRAM tr_cooling_logic (* task: 스캔 프로그램 *)
(* 온도 제어로 하절기 tr cooling fan 제어 *)
VAR
    temp_tr01_temp : WORD; (* temp_tr01_temp *)
    temp_tr02_temp : WORD; (* temp_tr02_temp *)
    temp_tr03_temp : WORD; (* temp_tr03_temp *)
    tr01_fan_operation AT M00212 : BIT;
    tr01_temp_high : BIT; (* tr01_temp_high *)
    tr01_temp_low : BIT; (* tr01_temp_low *)
    tr02_fan_operation AT M00213 : BIT;
    tr02_temp_high : BIT; (* tr02_temp_high *)
    tr02_temp_low : BIT; (* tr02_temp_low *)
    tr03_fan_operation AT M00214 : BIT;
    tr03_temp_high : BIT; (* tr03_temp_high *)
    tr03_temp_low : BIT; (* tr03_temp_low *)
    tr1_cooling_manual_start AT M00102 : BIT;
    tr2_cooling_manual_start AT M00103 : BIT;
    tr3_cooling_manual_start AT M00104 : BIT;
    tr_1_cooling_manual_out : BIT; (* tr_1_cooling_manual_out *)
    tr_1_cooling_out : BIT; (* tr_1_cooling_out *)
    tr_2_cooling_manual_out : BIT; (* tr_2_cooling_manual_out *)
    tr_2_cooling_out : BIT; (* tr_2_cooling_out *)
    tr_3_cooling_manual_out : BIT; (* tr_3_cooling_manual_out *)
    tr_3_cooling_out : BIT; (* tr_3_cooling_out *)
    tr_cooling_auto AT M00100 : BIT; (* tr_cooling_auto *)
    tr_cooling_start AT M00101 : BIT; (* tr_cooling_start *)
    tr_simulation_injection_temp_igh : WORD; (* tr_simulation_injection_temp_igh *)
    tr_simulation_injection_temp_low : WORD; (* tr_simulation_injection_temp_low *)
END_VAR
VAR_EXTERNAL
    tr01_1m_high_temp_from_pc : WORD; (* AT D00980 *)
    tr01_temp_scaled_value : WORD; (* AT D00024 *)
    tr02_1m_high_temp_from_pc : WORD; (* AT D00981 *)
    tr02_temp_scaled_value : WORD; (* AT D00025 *)
    tr03_1m_high_temp_from_pc : WORD; (* AT D00982 *)
    tr03_temp_scaled_value : WORD; (* AT D00026 *)
    _010_W_1hr_count : WORD; (* _010_W_1hr_count *)
    _010_W_TR1_temp_high_set : WORD; (* AT D00900 *)
    _010_W_TR1_temp_low_set : WORD; (* AT D00901 *)
    _010_W_TR2_temp_high_set : WORD; (* AT D00902 *)
    _010_W_TR2_temp_low_set : WORD; (* AT D00903 *)
    _010_W_TR3_temp_high_set : WORD; (* AT D00904 *) (* _010_W_TR_temp_high_set *)
    _010_W_TR3_temp_low_set : WORD; (* AT D00905 *) (* _010_W_TR_temp_low_set *)
    _01_CH0_TEMP : WORD; (* AT U01.04 *) (* 온도입력모듈 : 채널0 온도변환값(전기실온도) *)
    _01_CH1_TEMP : WORD; (* AT U01.05 *) (* 온도입력모듈 : 채널1 온도변환값(외기온도) *)
    _01_CH2_TEMP : WORD; (* AT U01.06 *) (* 온도입력모듈 : 채널2 온도변환값(에어콘01출구온도) *)
    _01_CH3_TEMP : WORD; (* AT U01.07 *) (* 온도입력모듈 : 채널3 온도변환값(에어콘02출구온도) *)
    _02_CH0_DATA : WORD; (* AT U02.02 *) (* 아날로그입력 모듈: 채널0 변환값(tr01 temp) *)
    _02_CH1_DATA : WORD; (* AT U02.03 *) (* 아날로그입력 모듈: 채널1 변환값(tr02 temp) *)
    _02_CH2_DATA : WORD; (* AT U02.04 *) (* 아날로그입력 모듈: 채널2 변환값(tr01 temp) *)
    월간타이머리셋 : BIT;
END_VAR
VAR_EXTERNAL RETAIN
    TR1_opertime_time : WORD;
    TR1_opertime_timer : TIMER;
    TR2_opertime_time : WORD;
    TR2_opertime_timer : TIMER;
    TR3_opertime_time : WORD;
    TR3_opertime_timer : TIMER;
    TR_opertime_total_time : WORD;
    _001_EF_tot_op_hour : WORD; (* _001_EF_tot_op_hour *)
    _001_SF_tot_op_hour : WORD; (* _001_SF_tot_op_hour *)
END_VAR

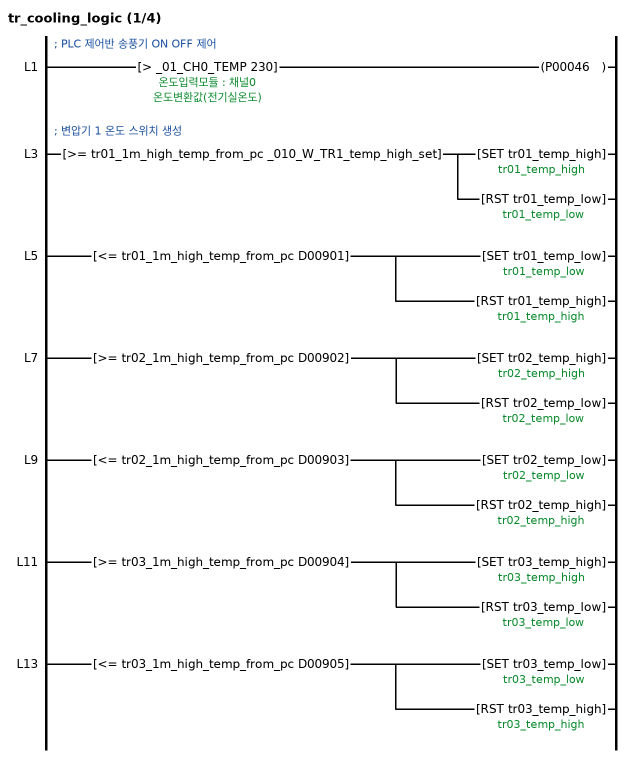
// PLC 제어반 송풍기 ON OFF 제어
; L1
LOAD>     _01_CH0_TEMP 230	// 온도입력모듈 : 채널0 온도변환값(전기실온도)
OUT       P00046
// 변압기 1 온도 스위치 생성
; L3
LOAD>=    tr01_1m_high_temp_from_pc _010_W_TR1_temp_high_set
SET       tr01_temp_high	// tr01_temp_high
RST       tr01_temp_low	// tr01_temp_low
; L5
LOAD<=    tr01_1m_high_temp_from_pc D00901
SET       tr01_temp_low	// tr01_temp_low
RST       tr01_temp_high	// tr01_temp_high
; L7
LOAD>=    tr02_1m_high_temp_from_pc D00902
SET       tr02_temp_high	// tr02_temp_high
RST       tr02_temp_low	// tr02_temp_low
; L9
LOAD<=    tr02_1m_high_temp_from_pc D00903
SET       tr02_temp_low	// tr02_temp_low
RST       tr02_temp_high	// tr02_temp_high
; L11
LOAD>=    tr03_1m_high_temp_from_pc D00904
SET       tr03_temp_high	// tr03_temp_high
RST       tr03_temp_low	// tr03_temp_low
; L13
LOAD<=    tr03_1m_high_temp_from_pc D00905
SET       tr03_temp_low	// tr03_temp_low
RST       tr03_temp_high	// tr03_temp_high

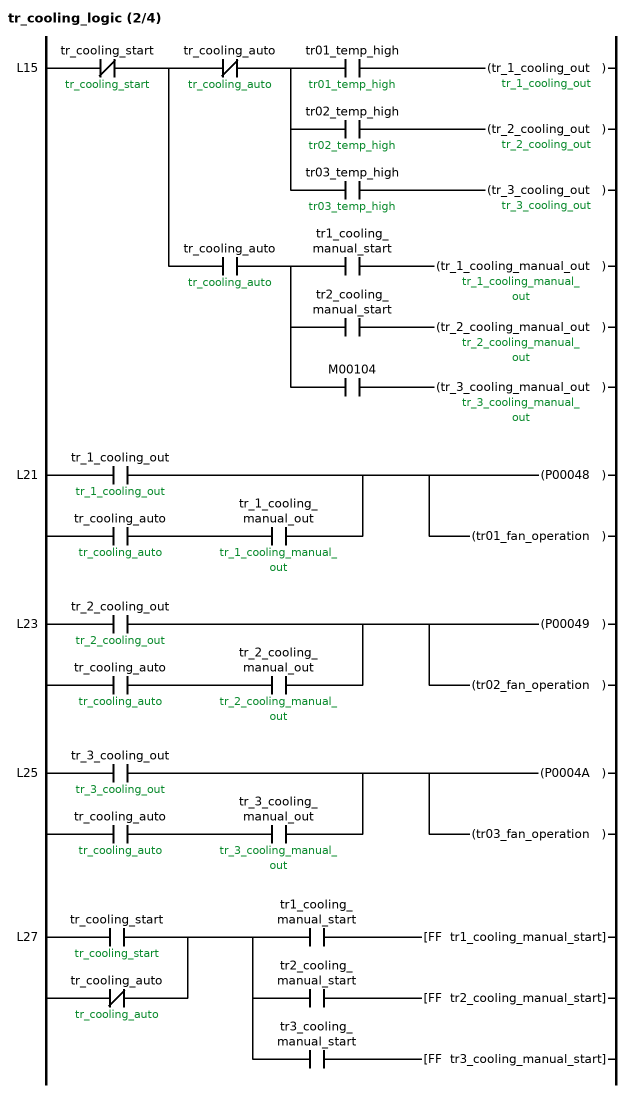
; L15
LOAD NOT  tr_cooling_start	// tr_cooling_start
MPUSH
AND NOT   tr_cooling_auto	// tr_cooling_auto
MPUSH
AND       tr01_temp_high	// tr01_temp_high
OUT       tr_1_cooling_out	// tr_1_cooling_out
MLOAD
AND       tr02_temp_high	// tr02_temp_high
OUT       tr_2_cooling_out	// tr_2_cooling_out
MPOP
AND       tr03_temp_high	// tr03_temp_high
OUT       tr_3_cooling_out	// tr_3_cooling_out
MPOP
AND       tr_cooling_auto	// tr_cooling_auto
MPUSH
AND       tr1_cooling_manual_start
OUT       tr_1_cooling_manual_out	// tr_1_cooling_manual_out
MLOAD
AND       tr2_cooling_manual_start
OUT       tr_2_cooling_manual_out	// tr_2_cooling_manual_out
MPOP
AND       M00104
OUT       tr_3_cooling_manual_out	// tr_3_cooling_manual_out
; L21
LOAD      tr_1_cooling_out	// tr_1_cooling_out
LOAD      tr_cooling_auto	// tr_cooling_auto
AND       tr_1_cooling_manual_out	// tr_1_cooling_manual_out
OR LOAD
OUT       P00048
OUT       tr01_fan_operation
; L23
LOAD      tr_2_cooling_out	// tr_2_cooling_out
LOAD      tr_cooling_auto	// tr_cooling_auto
AND       tr_2_cooling_manual_out	// tr_2_cooling_manual_out
OR LOAD
OUT       P00049
OUT       tr02_fan_operation
; L25
LOAD      tr_3_cooling_out	// tr_3_cooling_out
LOAD      tr_cooling_auto	// tr_cooling_auto
AND       tr_3_cooling_manual_out	// tr_3_cooling_manual_out
OR LOAD
OUT       P0004A
OUT       tr03_fan_operation
; L27
LOAD      tr_cooling_start	// tr_cooling_start
OR NOT    tr_cooling_auto	// tr_cooling_auto
MPUSH
AND       tr1_cooling_manual_start
FF        tr1_cooling_manual_start
MLOAD
AND       tr2_cooling_manual_start
FF        tr2_cooling_manual_start
MPOP
AND       tr3_cooling_manual_start
FF        tr3_cooling_manual_start

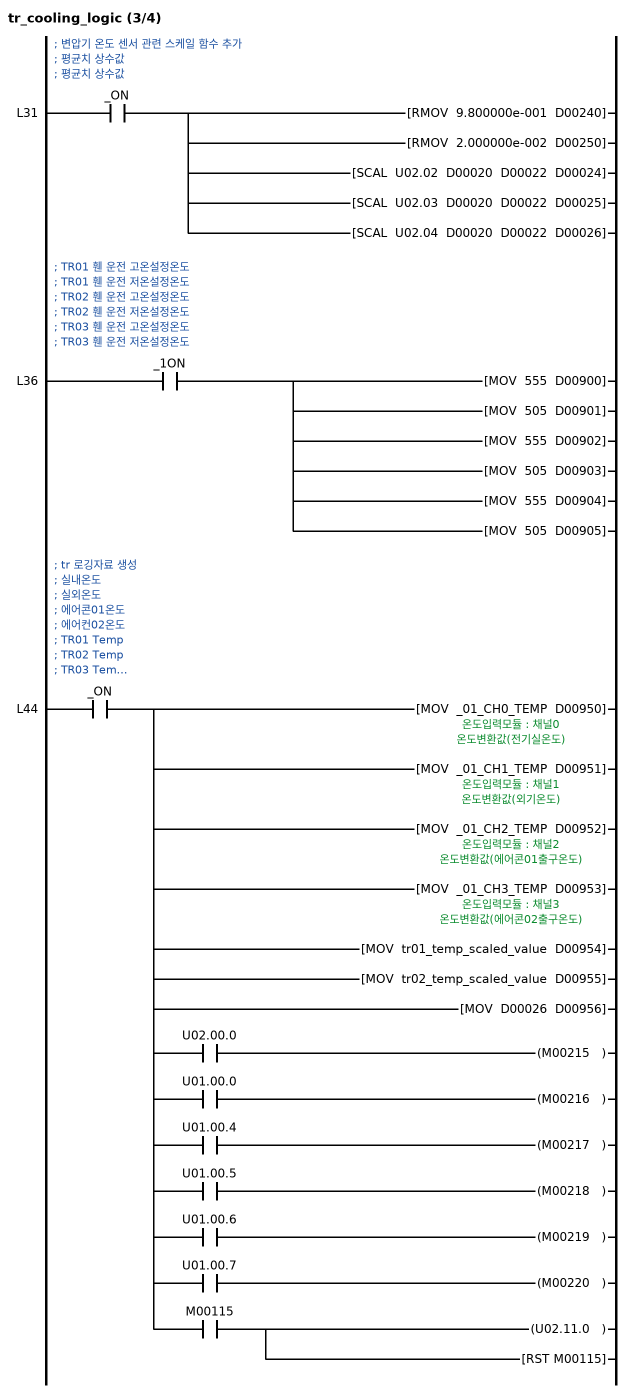
// 변압기 온도 센서 관련 스케일 함수 추가
; L31
LOAD      _ON
RMOV      9.800000e-001 D00240
RMOV      2.000000e-002 D00250
SCAL      U02.02 D00020 D00022 D00024
SCAL      U02.03 D00020 D00022 D00025
SCAL      U02.04 D00020 D00022 D00026
// output comment: 평균치 상수값
// output comment: 평균치 상수값
; L36
LOAD      _1ON
MOV       555 D00900
MOV       505 D00901
MOV       555 D00902
MOV       505 D00903
MOV       555 D00904
MOV       505 D00905
// output comment: TR01 휀 운전 고온설정온도
// output comment: TR01 휀 운전 저온설정온도
// output comment: TR02 휀 운전 고온설정온도
// output comment: TR02 휀 운전 저온설정온도
// output comment: TR03 휀 운전 고온설정온도
// output comment: TR03 휀 운전 저온설정온도
// tr 로깅자료 생성
; L44
LOAD      _ON
MOV       _01_CH0_TEMP D00950	// 온도입력모듈 : 채널0 온도변환값(전기실온도)
MOV       _01_CH1_TEMP D00951	// 온도입력모듈 : 채널1 온도변환값(외기온도)
MOV       _01_CH2_TEMP D00952	// 온도입력모듈 : 채널2 온도변환값(에어콘01출구온도)
MOV       _01_CH3_TEMP D00953	// 온도입력모듈 : 채널3 온도변환값(에어콘02출구온도)
MOV       tr01_temp_scaled_value D00954
MOV       tr02_temp_scaled_value D00955
MOV       D00026 D00956
MPUSH
AND       U02.00.0
OUT       M00215
MLOAD
AND       U01.00.0
OUT       M00216
MLOAD
AND       U01.00.4
OUT       M00217
MLOAD
AND       U01.00.5
OUT       M00218
MLOAD
AND       U01.00.6
OUT       M00219
MLOAD
AND       U01.00.7
OUT       M00220
MPOP
AND       M00115
OUT       U02.11.0
RST       M00115
// output comment: 실내온도
// output comment: 실외온도
// output comment: 에어콘01온도
// output comment: 에어컨02온도
// output comment: TR01 Temp
// output comment: TR02 Temp
// output comment: TR03 Temp
// output comment: 아날로그입력 모듈: 모듈 에러
// output comment: 온도입력모듈 : 모듈 에러
// output comment: 온도입력모듈 : 채널0 단선
// output comment: 온도입력모듈 : 채널1 단선 
// output comment: 온도입력모듈 : 채널2 단선
// output comment: 온도입력모듈 : 채널3 단선
// output comment: 입력모듈 오류 리셋 신호

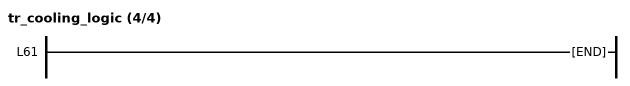
; L61
END
END_PROGRAM

PROGRAM initialzation (* task: init *)
(* 변수 초기값 입력 *)
VAR_EXTERNAL
    Park_1H_time : WORD;
    Park_manual_oper_time : WORD;
    Park_temp_1_high : WORD;
    Park_temp_1_high_H_set : WORD;
    Park_temp_1_high_L_set : WORD;
    Park_temp_2_med_high : WORD;
    Park_temp_2_med_high_H_set : WORD;
    Park_temp_2_med_high_L_set : WORD;
    Park_temp_3_med : WORD;
    Park_temp_3_med_H_set : WORD;
    Park_temp_3_med_L_set : WORD;
    Park_temp_4_med_low : WORD;
    Park_temp_4_med_low_H_set : WORD;
    Park_temp_4_med_low_L_set : WORD;
    Park_temp_5_low : WORD;
    Park_temp_5_low_H_set : WORD;
    Park_temp_5_low_L_set : WORD;
    Park_temp_6_low_1 : WORD;
    Park_temp_6_low_1_oper_time : WORD;
    Park_temp_7_low_2 : WORD;
    Park_temp_7_low_2_oper_time : WORD;
    Park_temp_8_low_3 : WORD;
    Park_temp_8_low_3_oper_time : WORD;
    Park_temp_9_below0 : WORD;
    Park_temp_9_below0_oper_time : WORD;
    Park_time_oper_delay_time : WORD;
    _007_outdoor_temp : WORD; (* _007_outdoor_temp *)
    _007_room_temp : WORD; (* _007_room_temp *)
    _008_room_temp_high_set : WORD; (* AT D00906 *) (* _008_room_temp_high_set *)
    _008_room_temp_high_set_high_limit : WORD; (* _008_room_temp_high_set_high_limit *)
    _008_room_temp_high_set_low_limit : WORD; (* _008_room_temp_high_set_low_limit *)
    _008_room_temp_low_set : WORD; (* AT D00907 *) (* _008_room_temp_low_set *)
    _008_room_temp_low_set_high_limit : WORD; (* _008_room_temp_low_set_high_limit *)
    _008_room_temp_low_set_low_limit : WORD; (* _008_room_temp_low_set_low_limit *)
    _009_outdoor_temp_high_set : WORD; (* AT D00908 *) (* _009_outdoor_temp_high_set *)
    _009_outdoor_temp_high_set_high_limit : WORD; (* _009_outdoor_temp_high_set_high_limit *)
    _009_outdoor_temp_high_set_low_limit : WORD; (* _009_outdoor_temp_high_set_low_limit *)
    _009_outdoor_temp_low_set : WORD; (* AT D00909 *) (* _009_outdoor_temp_low_set *)
    _009_outdoor_temp_low_set_high_limit : WORD; (* _009_outdoor_temp_low_set_high_limit *)
    _009_outdoor_temp_low_set_low_limit : WORD; (* _009_outdoor_temp_low_set_low_limit *)
    _010_W_1hr_count : WORD; (* _010_W_1hr_count *)
    _010_W_1_thousand_hour : WORD; (* _010_W_1_thousand_hour *)
    _010_W_fan_power_capacity : WORD; (* _010_W_fan_power_capacity *)
    _010_W_high_low_diff : WORD; (* _010_W_high_low_diff *)
    _010_W_power_unit_price : WORD; (* _010_W_power_unit_price *)
    주차장_급기가동온도 : WORD;
    주차장_급기정지온도 : WORD; (* 주차장_제어_외기_고온도 *)
END_VAR

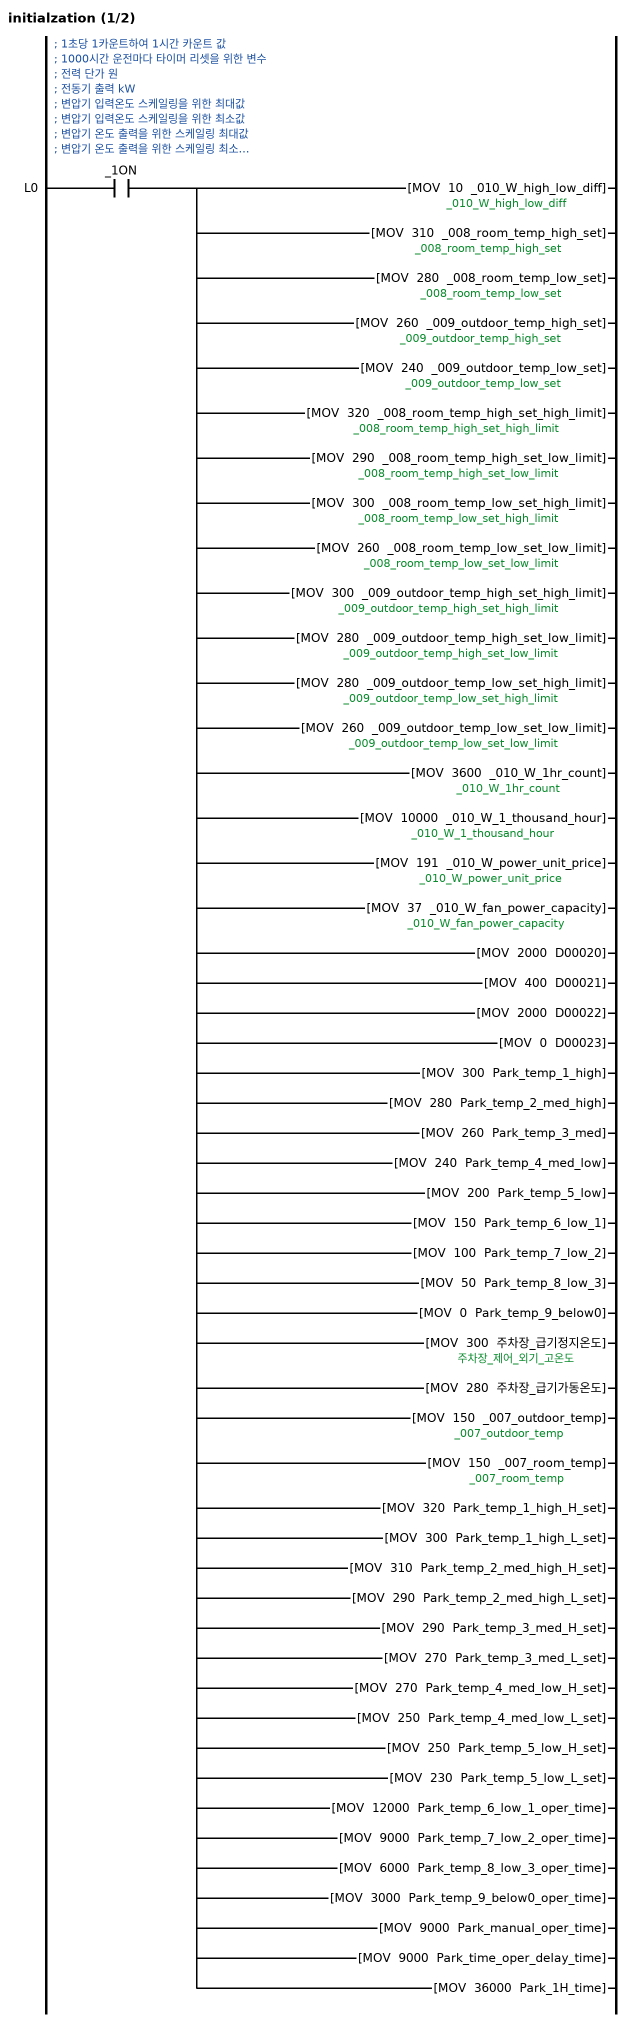
; L0
LOAD      _1ON
MOV       10 _010_W_high_low_diff	// _010_W_high_low_diff
MOV       310 _008_room_temp_high_set	// _008_room_temp_high_set
MOV       280 _008_room_temp_low_set	// _008_room_temp_low_set
MOV       260 _009_outdoor_temp_high_set	// _009_outdoor_temp_high_set
MOV       240 _009_outdoor_temp_low_set	// _009_outdoor_temp_low_set
MOV       320 _008_room_temp_high_set_high_limit	// _008_room_temp_high_set_high_limit
MOV       290 _008_room_temp_high_set_low_limit	// _008_room_temp_high_set_low_limit
MOV       300 _008_room_temp_low_set_high_limit	// _008_room_temp_low_set_high_limit
MOV       260 _008_room_temp_low_set_low_limit	// _008_room_temp_low_set_low_limit
MOV       300 _009_outdoor_temp_high_set_high_limit	// _009_outdoor_temp_high_set_high_limit
MOV       280 _009_outdoor_temp_high_set_low_limit	// _009_outdoor_temp_high_set_low_limit
MOV       280 _009_outdoor_temp_low_set_high_limit	// _009_outdoor_temp_low_set_high_limit
MOV       260 _009_outdoor_temp_low_set_low_limit	// _009_outdoor_temp_low_set_low_limit
MOV       3600 _010_W_1hr_count	// _010_W_1hr_count
MOV       10000 _010_W_1_thousand_hour	// _010_W_1_thousand_hour
MOV       191 _010_W_power_unit_price	// _010_W_power_unit_price
MOV       37 _010_W_fan_power_capacity	// _010_W_fan_power_capacity
MOV       2000 D00020
MOV       400 D00021
MOV       2000 D00022
MOV       0 D00023
MOV       300 Park_temp_1_high
MOV       280 Park_temp_2_med_high
MOV       260 Park_temp_3_med
MOV       240 Park_temp_4_med_low
MOV       200 Park_temp_5_low
MOV       150 Park_temp_6_low_1
MOV       100 Park_temp_7_low_2
MOV       50 Park_temp_8_low_3
MOV       0 Park_temp_9_below0
MOV       300 주차장_급기정지온도	// 주차장_제어_외기_고온도
MOV       280 주차장_급기가동온도
MOV       150 _007_outdoor_temp	// _007_outdoor_temp
MOV       150 _007_room_temp	// _007_room_temp
MOV       320 Park_temp_1_high_H_set
MOV       300 Park_temp_1_high_L_set
MOV       310 Park_temp_2_med_high_H_set
MOV       290 Park_temp_2_med_high_L_set
MOV       290 Park_temp_3_med_H_set
MOV       270 Park_temp_3_med_L_set
MOV       270 Park_temp_4_med_low_H_set
MOV       250 Park_temp_4_med_low_L_set
MOV       250 Park_temp_5_low_H_set
MOV       230 Park_temp_5_low_L_set
MOV       12000 Park_temp_6_low_1_oper_time
MOV       9000 Park_temp_7_low_2_oper_time
MOV       6000 Park_temp_8_low_3_oper_time
MOV       3000 Park_temp_9_below0_oper_time
MOV       9000 Park_manual_oper_time
MOV       9000 Park_time_oper_delay_time
MOV       36000 Park_1H_time
// output comment: 1초당 1카운트하여 1시간 카운트 값
// output comment: 1000시간 운전마다 타이머 리셋을 위한 변수
// output comment: 전력 단가 원
// output comment: 전동기 출력 kW
// output comment: 변압기 입력온도 스케일링을 위한 최대값
// output comment: 변압기 입력온도 스케일링을 위한 최소값
// output comment: 변압기 온도 출력을 위한 스케일링 최대값
// output comment: 변압기 온도 출력을 위한 스케일링 최소값
// output comment: 주차장 지역별 온도 제어를 위한 단계별 고설정치 및 저 설정치
// output comment: 주차장 시간운전 제어를 위한 운전 시간 초기값 입력
// output comment: 수동 시간운전 초기값 15분
// output comment: 온도 운전에서 시간운전 전환시 계속 운전 방지를 위한 지연시간 15분
// output comment: 1시간 주기운전을 위한 1시간 타이머 변수 입력

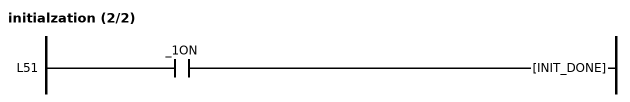
; L51
LOAD      _1ON
INIT_DONE
END_PROGRAM